{attribute 'linkalways'} 
{attribute 'no_explicit_call' := 'This FB is a CLASS and must be accessed using methods or properties'}
{attribute 'enable_dynamic_creation'}
FUNCTION_BLOCK Node_F_VN_RemapImageToPolarSpace EXTENDS VisionNode
VAR
    ipSrcImage : _ITcVnImage;
    ipDestImage : _ITcVnImage;
    aCenter : _TcVnPoint2_REAL;
    hrPrev : _HRESULT(S_OK);
	hresult : _HRESULT(S_OK);
END_VAR

METHOD PUBLIC  Clone : I_Node
VAR
	pNode : POINTER TO Node_F_VN_RemapImageToPolarSpace;
END_VAR
pNode := __NEW(Node_F_VN_RemapImageToPolarSpace);
Clone := pNode^;
END_METHOD

METHOD FB_init : BOOL
VAR_INPUT
	bInitRetains : BOOL; // if TRUE, the retain variables are initialized (warm start / cold start)
	bInCopyCode : BOOL;  // if TRUE, the instance afterwards gets moved into the copy code (online change)
END_VAR
AddInput('ipSrcImage', ipSrcImage);
AddInput('aCenter', aCenter);
AddInput('hrPrev', hrPrev);
AddOutput('ipDestImage', ipDestImage);
AddOutput('hresult',hresult);
END_METHOD

METHOD PROTECTED OnExecute
hresult.Value := F_VN_RemapImageToPolarSpace(
    ipSrcImage := ipSrcImage.Value,
	ipDestImage := ipDestImage.Value,
    aCenter := aCenter.Value,
	hrPrev:= hrPrev.Value);
END_METHOD

METHOD PUBLIC PreExecutionCheck
VAR_INPUT
	Check : I_PreExecutionChecks;
END_VAR
Check.IsTrue(ipSrcImage.IsValid, 'ipSrcImage must contain an image');
END_METHOD

END_FUNCTION_BLOCK

(* stored: Version 1.1.0.1, ProductVersion 3.1.4024.13
   POU Node_F_VN_RemapImageToPolarSpace: Id {8438fe45-4b8a-0f05-247e-af14d5118d5a}, SpecialFunc None
   Folder Constructor: Id {c0c918ff-f40e-0ddd-3c8b-7c69cd7f3f26}
   Method Clone: Id {ef20850c-22c5-02e3-24b7-bc9a7c394ec9}
   Method FB_init: Id {a11edaa2-f621-047a-02aa-acfea850d913}
   Method OnExecute: Id {96ad678f-1f48-0f6c-329a-0646dbb6db31}
   Method PreExecutionCheck: Id {e53c22d8-6595-038d-1496-473d2323c96e} *)
